{attribute 'qualified_only'}
{attribute 'strict'}
TYPE E_TL_Phase :
(
	INIT := 0,
	RED,
	GREEN,
	YELLOW,
	YELLOWRED
);
END_TYPE

(* stored: Version 1.1.0.1, ProductVersion 3.1.4024.12
   DUT E_TL_Phase: Id {4a04ad9d-b5ba-462a-8b8d-57ae1cd32cd1} *)
